// TIA Portal V20 export
// export: Created 2026-07-10T11:12:25.281741Z, ExportSetting WithDefaults, DisplayName Totally Integrated Automation Portal, DisplayVersion V20, DisplayName TIA Portal Openness, DisplayVersion V20, DisplayName TIA Portal Version Control Interface, DisplayVersion V20, DisplayName STEP 7 Professional, DisplayVersion V20, DisplayName STEP 7 Safety, DisplayVersion V20, DisplayName WinCC Basic/Comfort/Advanced, DisplayVersion V20, DisplayName WinCC Unified, DisplayVersion V20
FUNCTION_BLOCK "Alarms"   // FB17, SCL
{ S7_Optimized_Access := 'TRUE' }
VERSION : 0.1
// stored: AutoNumber true, IsIECCheckEnabled false, IsRetainMemResEnabled false, MemoryReserve 100, SetENOAutomatically false, UDAEnableTagReadback false
   VAR
      WaterOutMaxTON { S7_SetPoint := 'True'} : TON_TIME;
      WaterOutMinTON { S7_SetPoint := 'True'} : TON_TIME;
      WaterInMaxTON { S7_SetPoint := 'True'} : TON_TIME;
      WaterInMinTON { S7_SetPoint := 'True'} : TON_TIME;
      "step" { S7_SetPoint := 'True'} : Int;
      ChlorAlarm { S7_SetPoint := 'True'} : "ChlorConsumptionAlarm";
   END_VAR
BEGIN
   #step := 0;
   "MB".Table.Alarms_Open1:="AlarmOpen1";
   "MB".Table.Alarms_Open2:="AlarmOpen2";

   "MB".Table.Alarms_RCV1Max:="MB".Table.RCV1LevelValue>="MB".Table.LevelRCV1AlarmMax;
   "MB".Table.Alarms_RCV1Min:="MB".Table.RCV1LevelValue<="MB".Table.LevelRCV1AlarmMin;
   "MB".Table.Alarms_RCV2Max:="MB".Table.RCV2LevelValue>="MB".Table.LevelRCV2AlarmMax;
   "MB".Table.Alarms_RCV2Min:="MB".Table.RCV2LevelValue<="MB".Table.LevelRCV2AlarmMin;

   "MB".Table.Alarms_RCV1Error:="Inputs_DB".ErrorRCV1;
   "MB".Table.Alarms_RCV2Error:="Inputs_DB".ErrorRCV2;

   "MB".Table.Alarms_ChlorMax:="MB".Table.ChlorValue>="MB".Table.Chlor_ConcentAlarm;

   //"MB".Table.Alarms_NoFlow:= NOT("FlowSensor");

   "MB".Table.Alarms_NoPowerSupply:= NOT ("PowerSupply");

   #WaterOutMaxTON(IN := "MB".Table.WaterOutPressureValue >= "MB".Table.WaterOutMaxValue,
                   PT := "MB".Table.WaterOutAlarmTime * 1000);
   "MB".Table.Alarms_WaterOutMax := #WaterOutMaxTON.Q;

   #WaterOutMinTON(IN:="MB".Table.WaterOutPressureValue<="MB".Table.WaterOutMinValue,
                   PT:="MB".Table.WaterOutAlarmTime*1000);
   "MB".Table.Alarms_WaterOutMin := #WaterOutMinTON.Q;

   #WaterInMaxTON(IN:="MB".Table.WaterInPressureValue >= "MB".Table.WaterInPresMaxValue,
                  PT:="MB".Table.WaterInPresAlarmTime*1000);
   "MB".Table.Alarms_WaterInMax := #WaterInMaxTON.Q;

   #WaterInMinTON(IN:="MB".Table.WaterInPressureValue <= "MB".Table.WaterInPresMinValue,
                  PT:="MB".Table.WaterInPresAlarmTime*1000);

   #ChlorAlarm(HighAlarm=>"MB"  .Table.Alarms_ChlorLargeConsumption);


   "MB".Table.Alarms_WaterInMin := #WaterOutMinTON.Q;

   "SirenOut" := %DB1. > 0 AND NOT "MB".Table.HMI_SoundOff;
END_FUNCTION_BLOCK
